FUNCTION_BLOCK "Main"
VERSION : 0.1
   VAR_INPUT
      in1 : Bool;
   END_VAR

   VAR_OUTPUT
      out1 : Bool;
   END_VAR


BEGIN
NETWORK
TITLE =
      CLR;
      O #in1;
      ON #in1;
      = #out1;
      CALL "__CPROVER_assert"
      (  condition := #out1
      );

END_FUNCTION_BLOCK

